TYPE "PosFbk_ITF"
VERSION : 0.1
// Block: PosFbk_ITF
   STRUCT
      Sts : Struct
         Error : Bool;
         ErrorNotSynched : Bool;
         PresetAck : Bool;
         EncIsAbsolute : Bool;
         Position : LReal;
      END_STRUCT;
      Ctrl : Struct
         Rst : Bool;
         PresetCmd : Bool;
         PresetPosition : LReal;
      END_STRUCT;
   END_STRUCT;

END_TYPE
